(* PLC project bounded_scale, Dassault Systèmes ControlBuild 2024x *)
(* stored: creationDateTime 2023-10-03T11:13:32-01:00 *)

(* This module simulates a scaling equation. Form of the scaling equation is y = k (ax + b). *)
FUNCTION_BLOCK equipment_library.bounded_scale
  VAR_INPUT
    inputValue : REAL := 0.0;
  END_VAR
  VAR_OUTPUT
    realValue : REAL := 0.0;
    dintValue : DINT := 0;
    intValue : INT := 0;
  END_VAR
  VAR
    a : REAL := 0.0;
    b : REAL := 0.0;
    k : REAL := 0.0;
  END_VAR
  VAR CONSTANT
    minInput : REAL := 0.0;
    maxInput : REAL := 100.0;
    minOutput : REAL := 0.0;
    maxOutput : REAL := 100.0;
  END_VAR
  VAR
    d_scale : BOOL := false;
    v_d_scale : REAL := 0.0;
  END_VAR


ACTION C_source_code:
/* ----------------------------------------------------------------	*/
/* Type : Model of Operative Behaviour					*/
/* Category :  Toolbox							*/
/* Author : Dassault Systemes						*/
/* Update date : June 2018						*/
/* ----------------------------------------------------------------	*/
/* This module simulates the scaling of real variables			*/
/*	from bounded inputs and outputs.					*/
/* Form of the scaling equation is y = k (ax + b).			*/
/* ----------------------------------------------------------------	*/

if (d_scale) realValue = v_d_scale;
else {
	k = maxInput-minInput;
	if ( k != 0 ) {
		/* Calcul des coefficients de mise à l'échelle */
		a = ( maxOutput - minOutput );
		b = (( minOutput * maxInput ) - ( minInput * maxOutput ));

		/* Mise à l'échelle	*/
		realValue = 1/k * (( a * inputValue ) + b );
		if ( inputValue >= maxInput ) realValue = maxOutput;              
		if ( inputValue <= minInput ) realValue = minOutput;
		}
	else realValue = k;
	}

dintValue = realValue;

if ((dintValue >= -32768) && (dintValue <= 32767)) intValue = dintValue ;
else intValue  = 0;
END_ACTION
END_FUNCTION_BLOCK
